FUNCTION_BLOCK Revezamento_3_Motores_ok_HMI (* Service Interface Function Block Type *)
  (* Standard: 61499-2 *)
  (* Version 0.0, 25/02/2026, template *)
  PACKAGE Hidryco.HidrycoLib;
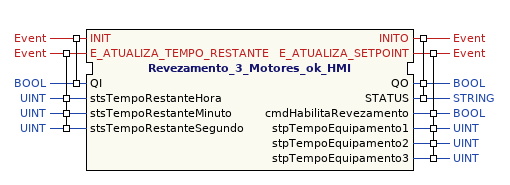
  EVENT_INPUT
    INIT WITH QI;
    E_ATUALIZA_TEMPO_RESTANTE WITH stsTempoRestanteHora, stsTempoRestanteMinuto, stsTempoRestanteSegundo;
  END_EVENT
  EVENT_OUTPUT
    INITO WITH QO, STATUS;
    E_ATUALIZA_SETPOINT WITH cmdHabilitaRevezamento, stpTempoEquipamento1, stpTempoEquipamento2, stpTempoEquipamento3;
  END_EVENT
  VAR_INPUT
    QI : BOOL;
    stsTempoRestanteHora : UINT;
    stsTempoRestanteMinuto : UINT;
    stsTempoRestanteSegundo : UINT;
  END_VAR
  VAR_OUTPUT
    QO : BOOL; (* Event Output Qualifier *)
    STATUS : STRING; (* Service Status *)
    cmdHabilitaRevezamento : BOOL;
    stpTempoEquipamento1 : UINT;
    stpTempoEquipamento2 : UINT;
    stpTempoEquipamento3 : UINT;
  END_VAR
  SERVICE /
    SEQUENCE 
    END_SEQUENCE
  END_SERVICE
END_FUNCTION_BLOCK
